{attribute 'GeneratedUsingTerminal: EPP4374-0002-0016'}
{attribute addProperty BoxType "EPP4374-0002-0016"}
{attribute addProperty Id "AI_Inputs_Channel_1AT %I*AI_Inputs_Channel_A8DF64E310AI_Inputs_Channel_2AT %I*AI_Inputs_Channel_A8DF64E310AO_Outputs_Channel_3AT %Q*AO_Outputs_Channel_BA7EBB7C2AO_Outputs_Channel_4AT %Q*AO_Outputs_Channel_BA7EBB7C2WcStateAT %I*WcState_9091E0EB2InfoDataAT %I*InfoData_32EB74EA10"}
{attribute addProperty CRC "1647443709"}
{attribute addProperty Size "36"}
TYPE EPP4374_6231FEFD EXTENDS EtcSlaveTerminalBase_947E5A46 :
STRUCT
	{attribute addProperty Name "AI_Inputs_Channel_1"}
	AI_Inputs_Channel_1 : AI_Inputs_Channel_A8DF64E3;
	{attribute addProperty Name "AI_Inputs_Channel_2"}
	AI_Inputs_Channel_2 : AI_Inputs_Channel_A8DF64E3;
	{attribute addProperty Name "AO_Outputs_Channel_3"}
	AO_Outputs_Channel_3 : AO_Outputs_Channel_BA7EBB7C;
	{attribute addProperty Name "AO_Outputs_Channel_4"}
	AO_Outputs_Channel_4 : AO_Outputs_Channel_BA7EBB7C;
	{attribute addProperty Name "WcState"}
	WcState : WcState_9091E0EB;
	{attribute addProperty Name "InfoData"}
	InfoData : InfoData_32EB74EA;
END_STRUCT
END_TYPE

(* stored: Version 1.2.0.0, ProductVersion 3.1.4024.9
   DUT EPP4374_6231FEFD: Id {09ba1b59-1195-4a32-a2c0-b564a82bc92f} *)
